FUNCTION_BLOCK UXIntPointerComparer EXTENDS Object IMPLEMENTS IPointerComparer
VAR
	_ClassName : STRING := __POUNAME();
END_VAR

{attribute 'monitoring' := 'call'}
PROPERTY ClassName : STRING
GET
ClassName := _ClassName;
END_GET
END_PROPERTY

{attribute "object_name" := "Compare"}
METHOD Compare : COMPARISION_RESULT
VAR_INPUT
	left : PVOID;
	right : PVOID;
END_VAR
VAR
	leftPointer : POINTER TO __UXINT; 
	rightPointer : POINTER TO __UXINT; 
END_VAR
IF left = 0 AND right = 0 THEN
	Compare := COMPARISION_RESULT.FIRST_EQUAL_TO_SECOND;
	RETURN;
END_IF

IF left = 0 THEN
	Compare := COMPARISION_RESULT.FIRST_LESS_THAN_SECOND;
	RETURN;	
END_IF

IF right = 0 THEN
	Compare := COMPARISION_RESULT.FIRST_GREATER_THAN_SECOND;
	RETURN;	
END_IF

leftPointer := left;
rightPointer := right;

IF leftPointer^ < rightPointer^ THEN
	Compare := COMPARISION_RESULT.FIRST_LESS_THAN_SECOND;
ELSIF leftPointer^ > rightPointer^ THEN
	Compare := COMPARISION_RESULT.FIRST_GREATER_THAN_SECOND;
ELSE
	Compare := COMPARISION_RESULT.FIRST_EQUAL_TO_SECOND;	
END_IF
END_METHOD

{attribute 'monitoring' := 'call'}
PROPERTY Size : ULINT
GET
Size := XSIZEOF(THIS^);
END_GET
END_PROPERTY

END_FUNCTION_BLOCK

(* stored: Version 1.1.0.1
   POU UXIntPointerComparer: Id {46b094cf-0d83-43dd-8f55-8c90ddd9417a}, SpecialFunc None
   Property ClassName: Id {3d1e4338-d3e6-497c-97d6-0ac58f71bef5}
   Get Get: Id {db0bdfc1-7f8e-41fc-95ee-bc780c15b1fb}
   Method Compare: Id {498c52ad-f6a6-4d11-bc99-94b2aae0c28f}
   Property Size: Id {c22a5dd3-cc2f-4add-9882-6d92a2c4cbd4}
   Get Get: Id {d4a3c89b-4c62-4312-b780-03ae48821a97} *)
